SUBAPPLICATION logiBUS_QXA_FROM_SUBSCRIBE_OPC (* Digitaler Ausgang, gesteuert von einem lokal ueberwachten OPC-UA-Knoten (von einem ANDEREN Geraet per CLIENT_1_0 remote beschrieben) - 'SUB style': das Protokoll (AX_SUBSCRIBE_1) steckt IM Baustein selbst, nicht in der Resource des Geraets *)
  (* Standard: 61499-2; Description: Copyright (c) 2026 Meisterschulen am Ostbahnhof This program and the accompanying materials are made available under the terms of the Eclipse Public License 2.0 which is available at https://www.eclipse.org/legal/epl-2.0/ SPDX-License-Identifier: EPL-2.0 *)
  (* Version 1.0, 2026-09-02, Franz Höpfinger, Meisterschulen am Ostbahnhof, initial API and implementation and/or initial documentation *)
  PACKAGE MyLib::sys;
  IMPORT logiBUS::io::DQ::logiBUS_DO;
  IMPORT logiBUS::io::DQ::logiBUS_DO_S;
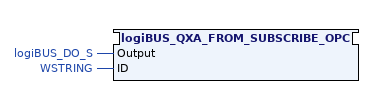
  VAR_INPUT
    Output : logiBUS::io::DQ::logiBUS_DO_S := logiBUS_DO::Invalid; (* Identify the Output Output_Q1..Q8 *)
    ID : WSTRING; (* Lokal ueberwachte Adresse (BOOL, ACTION=READ) - wird von einem anderen Geraet per CLIENT_1_0 remote beschrieben *)
  END_VAR
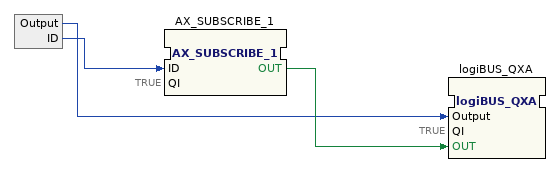
  FBS
    AX_SUBSCRIBE_1 : adapter::net::AX_SUBSCRIBE_1(QI := TRUE);
    logiBUS_QXA : logiBUS::io::DQ::logiBUS_QXA(QI := TRUE);
  END_FBS
  DATA_CONNECTIONS
    Output TO logiBUS_QXA.Output;
    ID TO AX_SUBSCRIBE_1.ID;
  END_CONNECTIONS
  ADAPTER_CONNECTIONS
    AX_SUBSCRIBE_1.OUT TO logiBUS_QXA.OUT;
  END_CONNECTIONS
END_SUBAPPLICATION
